(* IEC 61131-3 sources: SMART-IRRIGATION-OPTIMIZATION-SYSTEM/milestone2, 1 file *)

(* ---- SmartIrrigationV2.st ---- *)
(*SmartIrrigationV2.st
 * ST (IEC 61131-3) Implementation for Smart Irrigation Optimization System
 * Milestone 2
*)

PROGRAM SmartIrrigationV2
  VAR
    status: STRING := 'Milestone 2';
  END_VAR

  (* Placeholder for Structured Text implementation *)
END_PROGRAM
